// TIA Portal V20 export
TYPE "UDT_Service_StepMedium"
   STRUCT
      command : Array[0..0] of DWord;   // 'Command' configuration of control modules for sequencer
      force : Array[0..0] of DWord;   // 'Force' configuration of control modules for sequencer
      check : Array[0..0] of DWord;   // 'Check' configuration of control modules for sequencer
      "or" : Array[0..0] of DWord;   // Logical 'OR' configuration of control modules for sequencer
   END_STRUCT;
   // command[0] := 16#FFFFFFFF;
   // force[0] := 16#FFFFFFFF;
   // check[0] := 16#FFFFFFFF;
   // "or"[0] := 16#FFFFFFFF;
END_TYPE
